// TIA Portal project "elev11_V15" (V15)

(* hardware
DEVICE "S7300/ET200M station_1"  S7-300 station
   slot 0: "Rail_0"  Rail  6ES7 390-1***0-0AA0
   slot 2: "PLC_1"  CPU 313C-2 DP  6ES7 313-6CF03-0AB0  V2.6
      slot 0: "MPI interface_1"  X1
      slot 1: "DP interface_1"  X2
      slot 2: "DI 16/DO 16_1"  DI16/DO16
      slot 4: "Count_1"  Counter
*)

// ===== PLC "PLC_1"  CPU 313C-2 DP =====

VAR_GLOBAL   // PLC tag table "Default tag table"
   "encoder" AT %I0.0 : Bool;
   "sensor1" AT %I0.3 : Bool;
   "motor up" AT %Q0.0 : Bool;
   "motor down" AT %Q0.1 : Bool;
   "marker" AT %M0.0 : Bool;
   "f1" AT %M0.1 : Bool;
   "f2" AT %M0.2 : Bool;
   "f3" AT %M0.3 : Bool;
   "f4" AT %M0.4 : Bool;
   "f5" AT %M0.5 : Bool;
   "f6" AT %M0.6 : Bool;
   "count(1)" AT %MW10 : Int;
   "count(2)" AT %MW12 : Int;
   "count(3)" AT %MW14 : Int;
   "count(4)" AT %MW16 : Int;
   "count(5)" AT %MW18 : Int;
   "count(6)" AT %MW20 : Int;
   "Hscounter" AT %MD120 : DInt;
   "flat1" AT %MW22 : Word;
   "flat2" AT %MW24 : Word;
   "flat3" AT %MW26 : Word;
   "flat4" AT %MW28 : Word;
   "flat5" AT %MW30 : Word;
   "flat6" AT %MW32 : Word;
   "s1" AT %M3.1 : Bool;
   "s2" AT %M3.2 : Bool;
   "s3" AT %M3.3 : Bool;
   "s4" AT %M3.4 : Bool;
   "s5" AT %M3.5 : Bool;
   "Tag_3" AT %MW34 : Int;
   "s6" AT %M3.6 : Bool;
   "flat0" AT %M1.0 : Bool;
   "flat(1)" AT %M1.1 : Bool;
   "flat(2)" AT %M1.2 : Bool;
   "flat(3)" AT %M1.3 : Bool;
   "flat(4)" AT %M1.4 : Bool;
   "flat(5)" AT %M1.5 : Bool;
   "flat(6)" AT %M1.6 : Bool;
   "Tag_2" AT %M1.7 : Bool;
   "Tag_4" AT %MD40 : Time;
   "fe(0)" AT %M4.0 : Bool;
   "fe(1)" AT %M4.1 : Bool;
   "fe(2)" AT %M4.2 : Bool;
   "fe(3)" AT %M4.3 : Bool;
   "fe(4)" AT %M4.4 : Bool;
   "fe(5)" AT %M4.5 : Bool;
   "fe(6)" AT %M4.6 : Bool;
   "flat.e(0)" AT %M5.0 : Bool;
   "flat.e(1)" AT %M5.1 : Bool;
   "flat.e(2)" AT %M5.2 : Bool;
   "flat.e(3)" AT %M5.3 : Bool;
   "flat.e(4)" AT %M5.4 : Bool;
   "flat.e(5)" AT %M5.5 : Bool;
   "flat.e(6)" AT %M5.6 : Bool;
   "Tag_5" AT %MW36 : Int;
   "count.e(1)" AT %MW50 : Int;
   "count.e(2)" AT %MW52 : Int;
   "count.e(3)" AT %MW54 : Int;
   "count.e(4)" AT %MW56 : Int;
   "count.e(5)" AT %MW58 : Int;
   "count.e(6)" AT %MW60 : Int;
   "Tag_6" AT %ID1000 : DWord;
   "tag7" AT %MD124 : DInt;
   "Tag_7" AT %MD128 : DInt;
   "Tag_8" AT %MD132 : DInt;
   "Tag_9" AT %M6.0 : Bool;
   "Tag_10" AT %M6.1 : Bool;
   "Tag_11" AT %M6.2 : Bool;
   "Tag_12" AT %M6.3 : Bool;
   "Tag_13" AT %M6.4 : Bool;
   "Tag_14" AT %M6.5 : Bool;
   "Tag_15" AT %M6.6 : Bool;
   "Tag_16" AT %M7.1 : Bool;
   "Tag_17" AT %M7.2 : Bool;
   "Tag_18" AT %M7.3 : Bool;
   "Tag_19" AT %M7.4 : Bool;
   "Tag_20" AT %M7.5 : Bool;
   "Tag_21" AT %M7.6 : Bool;
   "Tag_1" AT %MD28 : DInt;
   "Tag_22" AT %M2.7 : Bool;
   "Tag_23" AT %MW48 : Int;
   "Tag_24" AT %MD110 : DInt;
   "Tag_25" AT %MW44 : Int;
   "int1" AT %M8.0 : Bool;
   "ext(1)" AT %M3.0 : Bool;
   "Tag_27" AT %M2.1 : Bool;
   "Tag_26" AT %M100.1 : Bool;
   "Tag_28" AT %M8.6 : Bool;
   "Tag_29" AT %M100.2 : Bool;
   "mw80" AT %MW80 : Word;
   "mw90" AT %MW90 : Int;
   "mw70" AT %MW38 : Int;
   "Tag_30" AT %M60.0 : Bool;
   "uppp" AT %M60.2 : Bool;
   "downn" AT %M60.3 : Bool;
   "Tag_31" AT %MD160 : DInt;
END_VAR

FUNCTION "FP" : Void   // FC1, SCL
{ S7_Optimized_Access := 'FALSE' }
VERSION : 0.1
   VAR_INPUT
      IN : Bool;
   END_VAR
   VAR_OUTPUT
      OUT : Bool;
   END_VAR
   VAR_IN_OUT
      Y : Bool;
   END_VAR
BEGIN
   #OUT := #IN AND NOT #Y;
   #Y := #IN;
END_FUNCTION

FUNCTION "FN" : Void   // FC2, SCL
{ S7_Optimized_Access := 'FALSE' }
VERSION : 0.1
   VAR_INPUT
      IN : Bool;
   END_VAR
   VAR_OUTPUT
      OUT : Bool;
   END_VAR
   VAR_IN_OUT
      X : Bool;
   END_VAR
BEGIN
   #OUT := NOT #IN AND #X;
   #X := #IN;
END_FUNCTION

FUNCTION "Block_1" : Void   // FC3, STL
{ S7_Optimized_Access := 'FALSE' }
VERSION : 0.1
BEGIN

REGION Network 1
         A(;
         O(;
         L     "Tag_8";
         L     DINT#120;
         ==D;
         );
         O(;
         L     "Tag_8";
         L     DINT#260;
         ==D;
         );
         O(;
         L     "Tag_8";
         L     DINT#440;
         ==D;
         );
         O(;
         L     "Tag_8";
         L     DINT#560;
         ==D;
         );
         O(;
         L     "Tag_8";
         L     DINT#710;
         ==D;
         );
         O(;
         L     "Tag_8";
         L     DINT#720;
         ==D;
         );
         );
         =     %L0.0;
         BLD   103;
         A(;
         O(;
         L     "Tag_8";
         L     DINT#-720;
         ==D;
         );
         O(;
         L     "Tag_8";
         L     DINT#-710;
         ==D;
         );
         O(;
         L     "Tag_8";
         L     DINT#-560;
         ==D;
         );
         O(;
         L     "Tag_8";
         L     DINT#-440;
         ==D;
         );
         O(;
         L     "Tag_8";
         L     DINT#-260;
         ==D;
         );
         O(;
         L     "Tag_8";
         L     DINT#-120;
         ==D;
         );
         );
         =     %L0.1;
         BLD   103;
         A     "sensor1";
         =     %L0.2;
         BLD   103;
         CALL  CTUD , "IEC_Counter_0_DB_2"
         ( CU := %L0.0,
           CD := %L0.1,
           R  := %L0.2,
           LD := ,
           PV := ,
           QU := ,
           QD := ,
           CV := "Tag_3"
         );
         NOP   0;
END_REGION

REGION Network 2
         L     0;
         L     "Tag_3";
         -I;
         T     "count(1)";
         NOP   0;
END_REGION

REGION Network 3
         A     "flat(1)";
         A(;
         L     "count(1)";
         L     0;
         <I;
         );
         AN    "uppp";
         AN    "flat(2)";
         AN    "flat(3)";
         AN    "flat(4)";
         AN    "flat(5)";
         AN    "Tag_22";
         S     "motor down";
END_REGION

REGION Network 4
         A     "flat(1)";
         A     "sensor1";
         R     "motor down";
END_REGION

REGION Network 5
         L     1;
         L     "Tag_3";
         -I;
         T     "count(2)";
         NOP   0;
END_REGION

REGION Network 6
         A     "flat(2)";
         A(;
         L     "count(2)";
         L     0;
         >I;
         );
         AN    "flat(1)";
         AN    "Tag_22";
         S     "motor up";
END_REGION

REGION Network 7
         A     "flat(2)";
         A(;
         L     "count(2)";
         L     0;
         <I;
         );
         AN    "flat(6)";
         AN    "flat(5)";
         AN    "flat(4)";
         AN    "flat(3)";
         AN    "uppp";
         AN    "Tag_22";
         S     "motor down";
END_REGION

REGION Network 8
         A     "flat(2)";
         A     "s1";
         R     "motor down";
         R     "motor up";
END_REGION

REGION Network 9
         L     2;
         L     "Tag_3";
         -I;
         T     "count(3)";
         NOP   0;
END_REGION

REGION Network 10
         A     "flat(3)";
         A(;
         L     "count(3)";
         L     0;
         >I;
         );
         AN    "flat(1)";
         AN    "flat(2)";
         AN    "Tag_22";
         S     "motor up";
END_REGION

REGION Network 11
         A     "flat(3)";
         A(;
         L     "count(3)";
         L     0;
         <I;
         );
         AN    "flat(6)";
         AN    "flat(5)";
         AN    "flat(4)";
         AN    "Tag_22";
         S     "motor down";
END_REGION

REGION Network 12
         A     "flat(3)";
         A     "s2";
         R     "motor down";
         R     "motor up";
END_REGION

REGION Network 13
         L     3;
         L     "Tag_3";
         -I;
         T     "count(4)";
         NOP   0;
END_REGION

REGION Network 14
         A     "flat(4)";
         A(;
         L     "count(4)";
         L     0;
         >I;
         );
         AN    "flat(1)";
         AN    "flat(2)";
         AN    "flat(3)";
         AN    "Tag_22";
         S     "motor up";
END_REGION

REGION Network 15
         A     "flat(4)";
         A(;
         L     "count(4)";
         L     0;
         <I;
         );
         AN    "flat(6)";
         AN    "flat(5)";
         AN    "Tag_22";
         S     "motor down";
END_REGION

REGION Network 16
         A     "flat(4)";
         A     "s3";
         R     "motor down";
         R     "motor up";
END_REGION

REGION Network 17
         L     4;
         L     "Tag_3";
         -I;
         T     "count(5)";
         NOP   0;
END_REGION

REGION Network 18
         A     "flat(5)";
         A(;
         L     "count(5)";
         L     0;
         >I;
         );
         AN    "flat(1)";
         AN    "flat(2)";
         AN    "flat(3)";
         AN    "flat(4)";
         AN    "Tag_22";
         S     "motor up";
END_REGION

REGION Network 19
         A     "flat(5)";
         A(;
         L     "count(5)";
         L     0;
         <I;
         );
         AN    "flat(6)";
         AN    "Tag_22";
         S     "motor down";
END_REGION

REGION Network 20
         A     "flat(5)";
         A     "s4";
         R     "motor down";
         R     "motor up";
END_REGION

REGION Network 21
         L     5;
         L     "Tag_3";
         -I;
         T     "count(6)";
         NOP   0;
END_REGION

REGION Network 22
         A     "flat(6)";
         A(;
         L     "count(6)";
         L     0;
         >I;
         );
         AN    "flat(1)";
         AN    "flat(2)";
         AN    "flat(3)";
         AN    "flat(4)";
         AN    "flat(5)";
         AN    "Tag_22";
         S     "motor up";
END_REGION

REGION Network 23
         A     "flat(6)";
         A(;
         L     "count(6)";
         L     0;
         <I;
         );
         AN    "Tag_22";
         S     "motor down";
END_REGION

REGION Network 24
         A     "flat(6)";
         A     "s5";
         R     "motor up";
END_REGION
END_FUNCTION

FUNCTION "extt" : Void   // FC4, STL
{ S7_Optimized_Access := 'FALSE' }
VERSION : 0.1
BEGIN

REGION Network 1
         A(;
         O(;
         L     "Tag_8";
         L     DINT#120;
         ==D;
         );
         O(;
         L     "Tag_8";
         L     DINT#260;
         ==D;
         );
         O(;
         L     "Tag_8";
         L     DINT#440;
         ==D;
         );
         O(;
         L     "Tag_8";
         L     DINT#560;
         ==D;
         );
         O(;
         L     "Tag_8";
         L     DINT#710;
         ==D;
         );
         O(;
         L     "Tag_8";
         L     DINT#720;
         ==D;
         );
         );
         =     %L0.0;
         BLD   103;
         A(;
         O(;
         L     "Tag_8";
         L     DINT#-720;
         ==D;
         );
         O(;
         L     "Tag_8";
         L     DINT#-710;
         ==D;
         );
         O(;
         L     "Tag_8";
         L     DINT#-560;
         ==D;
         );
         O(;
         L     "Tag_8";
         L     DINT#-440;
         ==D;
         );
         O(;
         L     "Tag_8";
         L     DINT#-260;
         ==D;
         );
         O(;
         L     "Tag_8";
         L     DINT#-120;
         ==D;
         );
         );
         =     %L0.1;
         BLD   103;
         A     "sensor1";
         =     %L0.2;
         BLD   103;
         CALL  CTUD , "IEC_Counter_0_DB"
         ( CU := %L0.0,
           CD := %L0.1,
           R  := %L0.2,
           LD := ,
           PV := ,
           QU := ,
           QD := ,
           CV := "Tag_5"
         );
         NOP   0;
END_REGION

REGION Network 2
         L     0;
         L     "Tag_5";
         -I;
         T     "count.e(1)";
         NOP   0;
END_REGION

REGION Network 3
         A     "flat.e(1)";
         A(;
         L     "count.e(1)";
         L     0;
         <I;
         );
         A     "int1";
         AN    "sensor1";
         AN    "flat.e(2)";
         AN    "flat.e(3)";
         AN    "flat.e(4)";
         AN    "flat.e(5)";
         AN    "flat.e(6)";
         S     "motor down";
END_REGION

REGION Network 4
         A     "sensor1";
         A     "flat.e(1)";
         A     "int1";
         R     "motor down";
END_REGION

REGION Network 5
         L     1;
         L     "Tag_5";
         -I;
         T     "count.e(2)";
         NOP   0;
END_REGION

REGION Network 6
         A     "flat.e(2)";
         A(;
         L     "count.e(2)";
         L     0;
         >I;
         );
         AN    "s1";
         AN    "flat.e(1)";
         AN    "flat.e(5)";
         A     "int1";
         S     "motor up";
END_REGION

REGION Network 7
         A     "flat.e(2)";
         A(;
         L     "count.e(2)";
         L     0;
         <I;
         );
         A     "int1";
         AN    "flat.e(6)";
         AN    "flat.e(5)";
         AN    "flat.e(4)";
         AN    "flat.e(3)";
         S     "motor down";
END_REGION

REGION Network 8
         A     "s1";
         A     "flat.e(2)";
         A     "int1";
         R     "motor down";
         R     "motor up";
END_REGION

REGION Network 9
         L     2;
         L     "Tag_5";
         -I;
         T     "count.e(3)";
         NOP   0;
END_REGION

REGION Network 10
         A     "flat.e(3)";
         A(;
         L     "count.e(3)";
         L     0;
         >I;
         );
         AN    "s2";
         AN    "flat.e(5)";
         A     "int1";
         AN    "flat.e(1)";
         AN    "flat.e(2)";
         S     "motor up";
END_REGION

REGION Network 11
         A     "flat.e(3)";
         A(;
         L     "count.e(3)";
         L     0;
         <I;
         );
         A     "int1";
         AN    "s2";
         AN    "flat.e(6)";
         AN    "flat.e(5)";
         AN    "flat.e(4)";
         S     "motor down";
END_REGION

REGION Network 12
         A     "s2";
         A     "flat.e(3)";
         A     "int1";
         R     "motor down";
         R     "motor up";
END_REGION

REGION Network 13
         L     3;
         L     "Tag_5";
         -I;
         T     "count.e(4)";
         NOP   0;
END_REGION

REGION Network 14
         A     "flat.e(4)";
         A(;
         L     "count.e(4)";
         L     0;
         >I;
         );
         AN    "flat.e(6)";
         A     "int1";
         AN    "flat.e(1)";
         AN    "flat.e(2)";
         AN    "flat.e(3)";
         S     "motor up";
END_REGION

REGION Network 15
         A     "flat.e(4)";
         A(;
         L     "count.e(4)";
         L     0;
         <I;
         );
         AN    "s3";
         A     "int1";
         AN    "flat.e(6)";
         AN    "flat.e(5)";
         S     "motor down";
END_REGION

REGION Network 16
         A     "s3";
         A     "flat.e(4)";
         A     "int1";
         R     "motor down";
         R     "motor up";
END_REGION

REGION Network 17
         L     4;
         L     "Tag_5";
         -I;
         T     "count.e(5)";
         NOP   0;
END_REGION

REGION Network 18
         A     "flat.e(5)";
         A(;
         L     "count.e(5)";
         L     0;
         >I;
         );
         AN    "s4";
         A     "int1";
         AN    "flat.e(1)";
         AN    "flat.e(2)";
         AN    "flat.e(3)";
         AN    "flat.e(4)";
         S     "motor up";
END_REGION

REGION Network 19
         A     "flat.e(5)";
         A(;
         L     "count.e(5)";
         L     0;
         <I;
         );
         AN    "s4";
         A     "int1";
         AN    "flat.e(6)";
         S     "motor down";
END_REGION

REGION Network 20
         A     "s4";
         A     "flat.e(5)";
         A     "int1";
         R     "motor down";
         R     "motor up";
END_REGION

REGION Network 21
         L     5;
         L     "Tag_5";
         -I;
         T     "count.e(6)";
         NOP   0;
END_REGION

REGION Network 22
         A     "flat.e(6)";
         A(;
         L     "count.e(6)";
         L     0;
         >I;
         );
         A     "int1";
         S     "motor up";
END_REGION

REGION Network 23
         A     "s5";
         A     "flat.e(6)";
         A     "int1";
         R     "motor up";
END_REGION
END_FUNCTION

FUNCTION "Block_3" : Void   // FC5, STL
{ S7_Optimized_Access := 'FALSE' }
VERSION : 0.1
BEGIN

REGION Network 1
         A     "sensor1";
         BLD   100;
         FP    "Tag_28";
         =     "Tag_29";
END_REGION

REGION Network 2
         AN    "motor up";
         AN    "motor down";
         =     %L0.0;
         A     %L0.0;
         =     %L0.1;
         BLD   103;
         CALL  TON , "IEC_Timer_0_DB"
         ( IN := %L0.1,
           PT := T#3s,
           Q  := "Tag_2",
           ET := "Tag_4"
         );
         NOP   0;
         A     %L0.0;
         AN    "Tag_2";
         =     "Tag_22";
END_REGION

REGION Network 3
         A     "motor up";
         JNB   Label_0;
         L     "Hscounter";
         T     "tag7";
   Label_0:NOP   0;
END_REGION

REGION Network 4
         A     "motor down";
         JNB   Label_1;
         L     "Hscounter";
         T     "Tag_7";
   Label_1:NOP   0;
END_REGION

REGION Network 5
         L     "tag7";
         L     "Tag_7";
         -D;
         T     "Tag_8";
         NOP   0;
END_REGION

REGION Network 6
         A     "sensor1";
         =     %L0.0;
         A     %L0.0;
         JNB   Label_2;
         L     DINT#0;
         T     "Tag_8";
   Label_2:NOP   0;
         A     %L0.0;
         JNB   Label_3;
         L     DINT#0;
         T     "tag7";
   Label_3:NOP   0;
         A     %L0.0;
         JNB   Label_4;
         L     DINT#0;
         T     "Tag_7";
   Label_4:NOP   0;
END_REGION

REGION Network 7
         O(;
         L     "Tag_3";
         L     1;
         ==I;
         );
         O(;
         L     "Tag_5";
         L     1;
         ==I;
         );
         =     "s1";
END_REGION

REGION Network 8
         O(;
         L     "Tag_3";
         L     2;
         ==I;
         );
         O(;
         L     "Tag_5";
         L     2;
         ==I;
         );
         =     "s2";
END_REGION

REGION Network 9
         O(;
         L     "Tag_3";
         L     3;
         ==I;
         );
         O(;
         L     "Tag_5";
         L     3;
         ==I;
         );
         =     "s3";
END_REGION

REGION Network 10
         O(;
         L     "Tag_3";
         L     4;
         ==I;
         );
         O(;
         L     "Tag_5";
         L     4;
         ==I;
         );
         =     "s4";
END_REGION

REGION Network 11
         O(;
         L     "Tag_3";
         L     5;
         ==I;
         );
         O(;
         L     "Tag_5";
         L     5;
         ==I;
         );
         =     "s5";
END_REGION

REGION Network 12
         O(;
         L     "Tag_3";
         L     6;
         ==I;
         );
         O(;
         L     "Tag_5";
         L     6;
         ==I;
         );
         =     "s6";
END_REGION

REGION Network 13
         A(;
         A     "fe(1)";
         BLD   100;
         FP    "Tag_16";
         );
         AN    "sensor1";
         S     "flat.e(1)";
END_REGION

REGION Network 14
         A     "sensor1";
         AN    "motor down";
         AN    "motor up";
         A     "Tag_2";
         A     "flat.e(1)";
         R     "flat.e(1)";
END_REGION

REGION Network 15
         A(;
         A     "fe(2)";
         BLD   100;
         FP    "Tag_17";
         );
         AN    "s1";
         S     "flat.e(2)";
END_REGION

REGION Network 16
         A     "s1";
         AN    "motor down";
         AN    "motor up";
         A     "Tag_2";
         A     "flat.e(2)";
         R     "flat.e(2)";
END_REGION

REGION Network 17
         A(;
         A     "fe(3)";
         BLD   100;
         FP    "Tag_18";
         );
         AN    "s2";
         S     "flat.e(3)";
END_REGION

REGION Network 18
         A     "s2";
         AN    "motor down";
         AN    "motor up";
         A     "Tag_2";
         A     "flat.e(3)";
         R     "flat.e(3)";
END_REGION

REGION Network 19
         A(;
         A     "fe(4)";
         BLD   100;
         FP    "Tag_19";
         );
         AN    "s3";
         S     "flat.e(4)";
END_REGION

REGION Network 20
         A     "s3";
         AN    "motor down";
         AN    "motor up";
         A     "Tag_2";
         A     "flat.e(4)";
         R     "flat.e(4)";
END_REGION

REGION Network 21
         A(;
         A     "fe(5)";
         BLD   100;
         FP    "Tag_20";
         );
         AN    "s4";
         S     "flat.e(5)";
END_REGION

REGION Network 22
         A     "s4";
         AN    "motor down";
         AN    "motor up";
         A     "Tag_2";
         A     "flat.e(5)";
         R     "flat.e(5)";
END_REGION

REGION Network 23
         A(;
         A     "fe(6)";
         BLD   100;
         FP    "Tag_21";
         );
         AN    "s5";
         S     "flat.e(6)";
END_REGION

REGION Network 24
         A     "s5";
         AN    "motor down";
         AN    "motor up";
         A     "Tag_2";
         A     "flat.e(6)";
         R     "flat.e(6)";
END_REGION

REGION Network 25
         A(;
         A     "f6";
         BLD   100;
         FP    "Tag_15";
         );
         AN    "s5";
         S     "flat(6)";
END_REGION

REGION Network 26
         A     "s5";
         AN    "motor down";
         AN    "motor up";
         A     "Tag_2";
         A     "flat(6)";
         R     "flat(6)";
END_REGION

REGION Network 27
         A(;
         A     "f5";
         BLD   100;
         FP    "Tag_14";
         );
         AN    "s4";
         S     "flat(5)";
END_REGION

REGION Network 28
         A     "s4";
         AN    "motor down";
         AN    "motor up";
         A     "Tag_2";
         A     "flat(5)";
         R     "flat(5)";
END_REGION

REGION Network 29
         A(;
         A     "f4";
         BLD   100;
         FP    "Tag_13";
         );
         AN    "s3";
         S     "flat(4)";
END_REGION

REGION Network 30
         A     "s3";
         AN    "motor down";
         AN    "motor up";
         A     "Tag_2";
         A     "flat(4)";
         R     "flat(4)";
END_REGION

REGION Network 31
         A(;
         A     "f3";
         BLD   100;
         FP    "Tag_12";
         );
         AN    "s2";
         S     "flat(3)";
END_REGION

REGION Network 32
         A     "s2";
         AN    "motor down";
         AN    "motor up";
         A     "Tag_2";
         A     "flat(3)";
         R     "flat(3)";
END_REGION

REGION Network 33
         A(;
         A     "f2";
         BLD   100;
         FP    "Tag_11";
         );
         AN    "s1";
         S     "flat(2)";
END_REGION

REGION Network 34
         A     "s1";
         AN    "motor down";
         AN    "motor up";
         A     "Tag_2";
         A     "flat(2)";
         R     "flat(2)";
END_REGION

REGION Network 35
         A(;
         A     "f1";
         BLD   100;
         FP    "Tag_10";
         );
         AN    "sensor1";
         S     "flat(1)";
END_REGION

REGION Network 36
         A     "sensor1";
         AN    "motor down";
         AN    "motor up";
         A     "Tag_2";
         A     "flat(1)";
         R     "flat(1)";
END_REGION

REGION Network 37
         AN    "flat.e(1)";
         AN    "flat.e(2)";
         AN    "flat.e(3)";
         AN    "flat.e(4)";
         AN    "flat.e(5)";
         AN    "flat.e(6)";
         =     "ext(1)";
END_REGION

REGION Network 38
         AN    "flat(1)";
         AN    "flat(2)";
         AN    "flat(3)";
         AN    "flat(4)";
         AN    "flat(5)";
         AN    "flat(6)";
         =     "int1";
END_REGION

REGION Network 39
         ON    "int1";
         ON    "ext(1)";
         S     "Tag_26";
END_REGION
END_FUNCTION

FUNCTION "Block_2" : Void   // FC7, STL
{ S7_Optimized_Access := 'FALSE' }
VERSION : 0.1
BEGIN

REGION Network 1
         AN    "sensor1";
         =     %L0.0;
         BLD   103;
         CALL  COUNT_300C , "COUNT_300C_DB"
         ( LADDR    := ,
           CHANNEL  := ,
           SW_GATE  := %L0.0,
           CTRL_DO  := ,
           SET_DO   := ,
           JOB_REQ  := ,
           JOB_ID   := ,
           JOB_VAL  := ,
           STS_GATE := ,
           STS_STRT := ,
           STS_LTCH := ,
           STS_DO   := ,
           STS_C_DN := ,
           STS_C_UP := ,
           COUNTVAL := "Hscounter",
           LATCHVAL := ,
           JOB_DONE := ,
           JOB_ERR  := ,
           JOB_STAT :=
         );
         NOP   0;
END_REGION

REGION Network 2
         AN    "Tag_26";
         S     "motor down";
END_REGION

REGION Network 3
         AN    "Tag_26";
         A     "sensor1";
         R     "motor down";
END_REGION
END_FUNCTION

ORGANIZATION_BLOCK "Main"   // OB1, SCL
TITLE = "Main Program Sweep (Cycle)"
{ S7_Optimized_Access := 'FALSE' }
VERSION : 0.1
   VAR_TEMP
      OB1_EV_CLASS : Byte;   // Bits 0-3 = 1 (Coming event), Bits 4-7 = 1 (Event class 1)
      OB1_SCAN_1 : Byte;   // 1 (Cold restart scan 1 of OB 1), 3 (Scan 2-n of OB 1)
      OB1_PRIORITY : Byte;   // Priority of OB Execution
      OB1_OB_NUMBR : Byte;   // 1 (Organization block 1, OB1)
      OB1_RESERVED_1 : Byte;   // Reserved for system
      OB1_RESERVED_2 : Byte;   // Reserved for system
      OB1_PREV_CYCLE : Int;   // Cycle time of previous OB1 scan (milliseconds)
      OB1_MIN_CYCLE : Int;   // Minimum cycle time of OB1 (milliseconds)
      OB1_MAX_CYCLE : Int;   // Maximum cycle time of OB1 (milliseconds)
      OB1_DATE_TIME : Date_And_Time;   // Date and time OB1 started
   END_VAR
BEGIN
   IF "sensor1"=1 THEN
       "motor down":=0
       ;
   END_IF;

   "Block_1"();
   "Block_2"();
   "extt"();
   "Block_3"();
END_ORGANIZATION_BLOCK

ORGANIZATION_BLOCK "COMPLETE RESTART"   // OB100, SCL
TITLE = "Complete Restart"
{ S7_Optimized_Access := 'FALSE' }
VERSION : 0.1
   VAR_TEMP
      OB100_EV_CLASS : Byte;   // 16#13, Event class 1, Entering event state, Event logged in diagnostic buffer
      OB100_STRTUP : Byte;   // 16#81/82/83/84 Method of startup
      OB100_PRIORITY : Byte;   // Priority of OB Execution
      OB100_OB_NUMBR : Byte;   // 100 (Organization block 100, OB100)
      OB100_RESERVED_1 : Byte;   // Reserved for system
      OB100_RESERVED_2 : Byte;   // Reserved for system
      OB100_STOP : Word;   // Event that caused CPU to stop (16#4xxx)
      OB100_STRT_INFO : DWord;   // Information on how system started
      OB100_DATE_TIME : Date_And_Time;   // Date and time OB100 started
   END_VAR
BEGIN
   IF "motor down"=0 THEN
       "motor down" := 1
       ;
   END_IF;
END_ORGANIZATION_BLOCK